// TwinCAT 3 PLC project Untitled1
// ProgramVersion: 3.1.4023.0
// libraries:
//   Tc2_Standard, * (Beckhoff Automation GmbH)
//   Tc2_System, * (Beckhoff Automation GmbH)
//   Tc3_Module, * (Beckhoff Automation GmbH)
// project tree:
//   / GlobalTextList.TcGTLO, PlcTask.TcTTO, Visualization Manager.TcVMO (not stored)
//   POUs/ MAIN.TcPOU
//   VISUs/ FILLER.TcVIS
// real-time tasks:
//   TASK PlcTask: cycle T#10ms, priority 20, ADS port 350

CONFIGURATION Untitled1
    RESOURCE PLC ON TwinCAT3
        TASK PlcTask(INTERVAL := T#10ms, PRIORITY := 20);
        PROGRAM MAIN WITH PlcTask : MAIN;
    END_RESOURCE
END_CONFIGURATION

// ---- POUs/MAIN.TcPOU
PROGRAM MAIN
VAR
	//outputs
	bConveyorMotor,bAutoLight,bManualLight,bInletValve:BOOL;
	
	//inputs
	bSensor1,bResetButton,bStopButton,bStartButton:BOOL;
	bSensor2,bSensor3:BOOL;
	bForwardButton,bReverseButton:BOOL;
	bLoadBottle, bRemoveBottle:BOOL;

	//triggers
	fbMyTrigger:r_trig;
	fbMyTrigger2:r_trig;
	
	//state variables
	bBottle1,bBottle2,bBottle3:BOOL; 
	bLiquidTank:BOOL;
	
	//States
	bForwardMode,bReverseMode:BOOL;
	bManualMode:BOOL;
	bAutoMode:BOOL;
	bOffMode:BOOL;
	
	//timers
	fbMyTimer:ton;
	fbMyTimer2:TON;
	fbMyTimer3:ton;
	fbMyTimer4:ton;
	
	//dints
	iTotalBottles:DINT;
	iState:DINT;
	iSelectorSwitch:DINT;
	iState2:UDINT;
	
	
	
	
	
	
END_VAR

//remember to see why it does not work in the case statement
IF bRemoveBottle THEN
		bRemoveBottle:=FALSE;
		bBottle3:=FALSE;
		bSensor3:=FALSE;						
		END_IF	

		
(*CASE iState2 OF
	0: IF bManualMode THEN
		iState2:=20;
		ELSIF bAutoMode THEN
			iState2:=10;
		END_IF
	10:	(*..................................AUTOMATIC MODE..............................................*)
				bManualMode:=FALSE;
				bAutoLight:=TRUE;
				bManualLight:=FALSE;
				//this is a state machine so we use CASE statement!
					IF bLoadBottle THEN
						bLoadBottle:=FALSE;
						bBottle1:=TRUE;
						IF bBottle1 THEN
							bSensor1:=TRUE;
					END_IF
				END_IF;
				
				IF bBottle1 AND NOT bBottle2 THEN
					bBottle1:=FALSE; bSensor1:=FALSE; bBottle2:=TRUE; //this simulates the conveyor!
				END_IF
	
				CASE iState OF
				0: IF bBottle2 THEN
					iState:=10;
					END_IF
				
				10: //we just got a bottle, let's fill it!
					IF  bBottle2 THEN 
						bSensor2:=TRUE;
						bInletValve:=TRUE;	
					END_IF
					fbMyTimer(in:=bBottle2,pt:=T#6S);
					IF fbMyTimer.Q THEN
						//bBottle2:=TRUE; //to change the color variable!
						bInletValve:=FALSE;
						fbMyTimer(in:=FALSE);
					
						iState:=20;
					END_IF
					
				20: //now we get the bottle of the conveyor
					IF bBottle2 AND NOT bBottle3 THEN
						bBottle2:=FALSE; bBottle3:=TRUE; bSensor2:=FALSE; bSensor3:=TRUE;
						iState:=30;
						END_IF
						 
				30: //we now want to count the number of bottles counted!
					iTotalBottles:=	iTotalBottles +1;
						iState:=0;
				END_CASE 
				
	20:
		(*..........................................MANUAL MODE............................................*)
				
									(*...................FORWARD DIRECTION...............*)
				bManualMode:=TRUE;
				bAutoLight:=FALSE;
				bManualLight:=TRUE;
				//this is a state machine so we use CASE statement!
					IF bForwardButton THEN
						bForwardButton:=FALSE;
						bBottle1:=TRUE;
						IF bBottle1 THEN
							bSensor1:=TRUE;
					END_IF
				END_IF;
				
				IF bBottle1 AND NOT bBottle2 THEN
					bBottle1:=FALSE; bSensor1:=FALSE; bBottle2:=TRUE; //this simulates the conveyor!
				END_IF
	
				CASE iState OF
				0: IF bBottle2 THEN
					iState:=10;
					END_IF
				
				10: //we just got a bottle, let's fill it!
					IF  bBottle2 THEN 
						bSensor2:=TRUE;
						//bInletValve:=TRUE;	
					END_IF
					fbMyTimer(in:=bInletValve,pt:=T#6S);
					IF fbMyTimer.Q THEN
						//bBottle2:=TRUE; //to change the color variable!
						bInletValve:=FALSE;
						fbMyTimer(in:=FALSE);
					
						iState:=20;
					END_IF
					
				20: //now we get the bottle of the conveyor
					IF bBottle2 AND NOT bBottle3 THEN
						bBottle2:=FALSE; bBottle3:=TRUE; bSensor2:=FALSE; bSensor3:=TRUE;
						iState:=30;
						END_IF
						 
				30: //we now want to count the number of bottles counted!
					iTotalBottles:=	iTotalBottles +1;
						iState:=0;
				END_CASE 
				
				
				
				(*...................................REVERSE DIRECTION...............................*)
				bManualMode:=TRUE;
				bAutoLight:=FALSE;
				bManualLight:=TRUE;
				//this is a state machine so we use CASE statement!
					IF bReverseButton THEN
						bReverseButton:=FALSE;
						bBottle3:=TRUE;
						IF bBottle3 THEN
							bSensor3:=TRUE;
					END_IF
				END_IF;
				
				IF bBottle3 AND NOT bBottle2 THEN
					bBottle3:=FALSE; bSensor3:=FALSE; bBottle2:=TRUE; //this simulates the conveyor!
				END_IF
	
				CASE iState OF
				0: IF bBottle2 THEN
					iState:=10;
					END_IF
				
				10: //we just got a bottle, let's fill it!
					IF  bBottle2 THEN 
						bSensor2:=TRUE;
						//bInletValve:=TRUE;	
					END_IF
					fbMyTimer(in:=bInletValve,pt:=T#6S);
					IF fbMyTimer.Q THEN
						//bBottle2:=TRUE; //to change the color variable!
						bInletValve:=FALSE;
						fbMyTimer(in:=FALSE);
					
						iState:=20;
					END_IF
					
				20: //now we get the bottle of the conveyor
					IF bBottle2 AND NOT bBottle1 THEN
						bBottle2:=FALSE; bBottle1:=TRUE; bSensor2:=FALSE; bSensor1:=TRUE;
						iState:=25;
						END_IF
						
				25: bBottle1:=FALSE;  bSensor1:=FALSE;
						
						iState:=30;
						 
				30: //we now want to count the number of bottles counted!
					iTotalBottles:=	iTotalBottles +1;
						iState:=0;
				END_CASE 
END_CASE*)
//IF bAutoMode THEN
//	bAutoMode:=FALSE;
//	bAutoLight:=TRUE; bManualMode:=FALSE; bManualLight:=FALSE;
	
//ELSIF bManualMode THEN
//			bManualMode:=FALSE; //like using an r_trig. always be careful with these!
//			bManualLight:=TRUE; bAutoLight:=FALSE; bAutoMode:=FALSE;
//END_IF		 

IF  bAutoMode THEN
				bManualLight:=FALSE;
				bManualMode:=FALSE;
				bAutoLight:=TRUE;
				//bAutoMode:=FALSE;
				
		//this is a state machine so we use CASE statement!
					IF bLoadBottle THEN
						bLoadBottle:=FALSE;
						bBottle1:=TRUE;
						IF bBottle1 THEN
							bSensor1:=TRUE;
					END_IF
				END_IF;
				
				IF bBottle1 AND NOT bBottle2 THEN
					bConveyorMotor:=TRUE;
					bSensor1:=TRUE;
					fbMyTimer4(in:=bBottle1,pt:=T#1S);
						IF fbMyTimer4.Q THEN
							fbMyTimer4(in:=FALSE);
								bBottle1:=FALSE; bSensor1:=FALSE; bBottle2:=TRUE; //this simulates the conveyor!					
							END_IF
				END_IF
				IF bStopButton THEN
					iState:=999;		
					bStopButton:=FALSE;							
				IF bResetButton THEN
					bAutoMode:=FALSE; 
					bBottle2:=FALSE;
					iState:=0;
					bResetButton:=FALSE;
					
				END_IF
		END_IF
				CASE iState OF
				0: IF bBottle2 THEN									
					iState:=10;
					END_IF
				
				10: //we just got a bottle, let's fill it!
					IF  bBottle2 THEN 
						bSensor2:=TRUE;
						bInletValve:=TRUE;	
					END_IF
					fbMyTimer(in:=bBottle2,pt:=T#2S);
					IF fbMyTimer.Q THEN
						//bBottle2:=TRUE; //to change the color variable!
						bInletValve:=FALSE;
						fbMyTimer(in:=FALSE);
					
						iState:=20;
					END_IF
					
				20: //now we get the bottle of the conveyor
					IF bBottle2 AND NOT bBottle3 THEN
						bBottle2:=FALSE; bBottle3:=TRUE; bSensor2:=FALSE; bSensor3:=TRUE;
						iState:=30;
						END_IF
						 
				30: //we now want to count the number of bottles counted!
					iTotalBottles:=	iTotalBottles +1;
						iState:=40;
						
				40:  fbMyTimer2(in:=bBottle3,pt:=T#998MS);
						IF fbMyTimer2.Q THEN
							fbMyTimer2(in:=FALSE);
							bBottle3:=FALSE;
							bSensor3:=FALSE;
							bBottle1:=TRUE;				
							iState:=10;
						END_IF
				END_CASE 
				
	
END_IF
(*.....note this commented endif is to try out the auto and man lights.....*)


IF bManualMode THEN
		bManualLight:=TRUE;
		bAutoLight:=FALSE;
		bAutoMode:=FALSE;
	
	IF bReverseMode THEN
		 
		bManualMode:=TRUE;
				bAutoLight:=FALSE;
				bManualLight:=TRUE;
				//this is a state machine so we use CASE statement!
					IF bReverseButton THEN
						//bReverseButton:=FALSE;
						bBottle3:=TRUE;
						IF bBottle3 THEN
							bSensor3:=TRUE;
					END_IF
				END_IF;
				
				IF bBottle3 AND NOT bBottle2 THEN
					bBottle3:=FALSE; bSensor3:=FALSE; bBottle2:=TRUE; //this simulates the conveyor!
				END_IF
	
				CASE iState OF
				0: IF bBottle2 THEN
					iState:=10;
					END_IF
				
				10: //we just got a bottle, let's fill it!
					IF  bBottle2 THEN 
						bSensor2:=TRUE;
						//bInletValve:=TRUE;	
					END_IF
					fbMyTimer(in:=bInletValve,pt:=T#6S);
					IF fbMyTimer.Q THEN
						//bBottle2:=TRUE; //to change the color variable!
						bInletValve:=FALSE;
						fbMyTimer(in:=FALSE);
					
						iState:=20;
					END_IF
					
				20: //now we get the bottle of the conveyor
					IF bBottle2 AND NOT bBottle1 THEN
						bBottle2:=FALSE; bBottle1:=TRUE; bSensor2:=FALSE; bSensor1:=TRUE;
						iState:=25;
						END_IF
						
				25: bBottle1:=FALSE;  bSensor1:=FALSE;
						
						iState:=30;
						 
				30: //we now want to count the number of bottles counted!
					iTotalBottles:=	iTotalBottles +1;
						iState:=0;
				END_CASE 
			bReverseMode:=FALSE;
		
		ELSIF bForwardMode THEN
				(*...................FORWARD DIRECTION...............*)
				IF bStopButton THEN
					bBottle3:=FALSE;
					bSensor3:=FALSE;
					bStopButton:=FALSE;							
						END_IF
			//bForwardMode:=FALSE;
				bManualMode:=TRUE;
				bAutoLight:=FALSE;
				bManualLight:=TRUE;
				//this is a state machine so we use CASE statement!
					IF bForwardButton THEN
						bForwardButton:=FALSE;
						bBottle1:=TRUE;
						IF bBottle1 THEN
							bSensor1:=TRUE;
					END_IF
				END_IF;
				IF bBottle1 AND NOT bBottle2 THEN
					bConveyorMotor:=TRUE;
					bSensor1:=TRUE;
					fbMyTimer4(in:=bBottle1,pt:=T#1S);
						IF fbMyTimer4.Q THEN
							fbMyTimer4(in:=FALSE);
								bBottle1:=FALSE; bSensor1:=FALSE; bBottle2:=TRUE; //this simulates the conveyor!					
							END_IF
				END_IF
				
//				IF bBottle1 AND NOT bBottle2 THEN
//					bBottle1:=FALSE; bSensor1:=FALSE; bBottle2:=TRUE; //this simulates the conveyor!
//				END_IF
	
				CASE iState OF
				0: IF bBottle2 THEN
					iState:=10;
					END_IF
				
				10: //we just got a bottle, let's fill it!
					IF  bBottle2 THEN 
						bSensor2:=TRUE;
						//bInletValve:=TRUE;	
					END_IF
					fbMyTimer(in:=bInletValve,pt:=T#2S);
					IF fbMyTimer.Q THEN
						//bBottle2:=TRUE; //to change the color variable!
						bInletValve:=FALSE;
						fbMyTimer(in:=FALSE);
					
						iState:=20;
					END_IF
					
				20: //now we get the bottle of the conveyor
					IF bBottle2 AND NOT bBottle3 THEN
						bBottle2:=FALSE; bBottle3:=TRUE; bSensor2:=FALSE; bSensor3:=TRUE;
						iState:=30;
						END_IF
						 
				30: //we now want to count the number of bottles counted!
					iTotalBottles:=	iTotalBottles +1;
						
						iState:=40;
						
				40:	fbMyTimer2(in:=bBottle3,pt:=T#998MS);
						IF fbMyTimer2.Q THEN
							fbMyTimer2(in:=FALSE);
							bBottle3:=FALSE;
							bSensor3:=FALSE;
							bBottle1:=TRUE;				
							iState:=10;
						END_IF
				END_CASE 
				
			
	END_IF
	
	
END_IF

END_PROGRAM

// ---- GlobalTextList.TcGTLO
TEXTLIST GlobalTextList
  795 = '<<<<'
  844 = '>>>>'
  3 = 'AUTO'
  646 = 'b1'
  984 = 'Bottle'
  243 = 'Bottle 1'
  992 = 'bottle 1'
  459 = 'bottle 2'
  172 = 'bottle 3'
  183 = 'CONVEYOR'
  698 = 'Elapsed Time %s'
  906 = 'Fanta'
  835 = 'FWD'
  762 = 'Inlet valve'
  905 = 'LIQUID TANK'
  407 = 'MAN'
  681 = 'MINI HMI'
  128 = 'REMOVE'
  934 = 'RST'
  408 = 'RVS'
  541 = 's1'
  350 = 's2'
  840 = 's3'
  671 = 'START'
  304 = 'STOP'
  975 = 'Total Bottles Filled: %d'
  451 = 'VALVE'
END_TEXTLIST

// ---- VISUs/FILLER.TcVIS
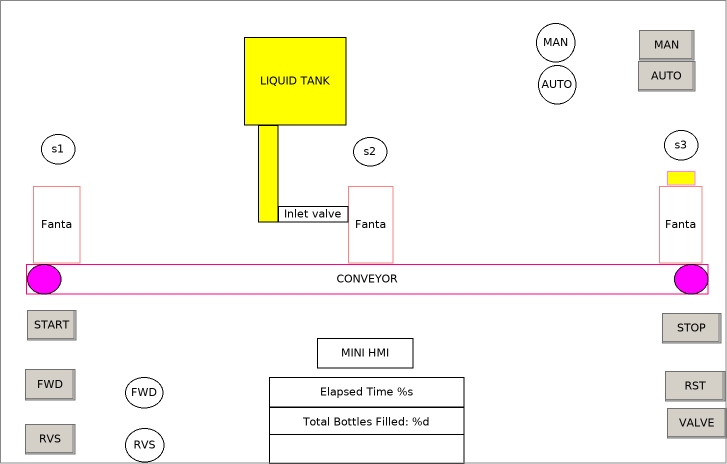
VISUALIZATION FILLER  // 727x464
    Ellipse (41,134 34x30), "s1", colour toggle: MAIN.bSensor1
    Ellipse (353,137 34x29), "s2", colour toggle: MAIN.bSensor2
    Ellipse (664,130 34x30), "s3", colour toggle: MAIN.bSensor3
    RoundedRectangle (33,186 47x77), "Fanta", invisible if: not MAIN.bBottle1
    RoundedRectangle (348,186 45x77), "Fanta", colour toggle: MAIN.bBottle2, invisible if: not MAIN.bBottle2
    RoundedRectangle (659,186 43x77), "Fanta", colour toggle: MAIN.bBottle3, invisible if: not MAIN.bBottle3
    Rectangle (244,37 102x88), "LIQUID TANK"
    Button (662,313 59x30), "STOP"
        OnMouseClick: execute { main.bStopButton:=TRUE; }
    Button (27,310 49x30), "START"
        OnMouseClick: execute { main.bLoadBottle:=true; }
    Button (638,61 57x30), "AUTO"
        OnMouseClick: execute { main.bAutoMode:=TRUE; }
    Button (639,30 55x30), "MAN"
        OnMouseClick: execute { main.bManualMode:=true; }
    Button (665,371 60x30), "RST"
        OnMouseClick: execute { main.bResetButton:=TRUE; }
    Button (667,408 60x30), "VALVE"
        OnMouseClick: execute { main.bInletValve:=TRUE; }
    Button (25,424 50x30), "RVS"
        OnMouseClick: execute { main.bReverseMode:=TRUE; main.bReverseButton:=TRUE; }
    Button (25,369 50x31), "FWD"
        OnMouseClick: execute { main.bForwardMode:=TRUE; main.bForwardButton:=TRUE; }
    Ellipse (536,23 39x39), "MAN", colour toggle: MAIN .bManualLight
    Ellipse (538,65 38x39), "AUTO", colour toggle: MAIN.bAutoLight
    Rectangle (269,377 195x30), "Elapsed Time %s", text variable: MAIN.fbMyTimer.ET
    Rectangle (269,407 195x30), "Total Bottles Filled: %d", text variable: MAIN.iTotalBottles
    Rectangle (269,434 195x30)
    RoundedRectangle (317,338 96x30), "MINI HMI"
    Rectangle (258,125 20x97)
    Rectangle (278,206 70x16), "Inlet valve", colour toggle: MAIN.bInletValve
    RoundedRectangle (26,264 682x30), "CONVEYOR", colour toggle: MAIN.bConveyorMotor
    Ellipse (674,264 34x30)
    Ellipse (27,264 34x30)
    Rectangle (667,171 28x14), invisible if: not MAIN.bBottle3
    Ellipse (125,377 38x31), "FWD", colour toggle: MAIN.bForwardMode
    Ellipse (125,428 39x34), "RVS", colour toggle: MAIN.bReverseMode
END_VISUALIZATION
